// TIA Portal V18 export
// export: Created 2026-06-08T04:47:36.6664765Z, ExportSetting WithDefaults, DisplayName Totally Integrated Automation Portal, DisplayVersion V18, DisplayName TIA Portal Openness, DisplayVersion V18, DisplayName TIA Portal Version Control Interface, DisplayVersion V18, DisplayName STEP 7 Professional, DisplayVersion V18, DisplayName STEP 7 Safety, DisplayVersion V18, DisplayName WinCC Professional, DisplayVersion V18
DATA_BLOCK "MB_SERVER_DB"   // DB53
// stored: AutoNumber true, DBAccessibleFromOPCUA true, InstanceOfName MB_SERVER_3, OfSystemLibElement MB_SERVER, OfSystemLibVersion 3.1
"MB_SERVER_3"
   // VAR_INPUT
   //    DISCONNECT : Bool;
   //    CONNECT_ID : UInt;
   //    IP_PORT : UInt;
   // END_VAR
   // VAR_OUTPUT
   //    NDR : Bool;
   //    DR : Bool;
   //    ERROR : Bool;
   //    STATUS : Word;
   // END_VAR
   // VAR_IN_OUT
   //    MB_HOLD_REG : Variant;
   // END_VAR
   // VAR
   //    TCON_SFB { S7_SetPoint := 'True'} : TCON;
   //    TDISCON_SFB { S7_SetPoint := 'True'} : TDISCON;
   //    TSEND_SFB { S7_SetPoint := 'True'} : TSEND;
   //    TRCV_SFB { S7_SetPoint := 'True'} : TRCV;
   //    TCON_Param { S7_SetPoint := 'True'} : TCON_Param;
   //    MB_State : UInt;
   //    Request_Count : UInt;
   //    Server_Message_Count : UInt;
   //    Xmt_Rcv_Count : UInt;
   //    Exception_Count : UInt;
   //    Success_Count : UInt;
   //    SL_Status_Hold : UInt;
   //    HR_Start_Offset : UInt;
   //    Init_OK : Bool;
   //    SL_Error_State : Bool;
   //    Connected : Bool;
   //    XMT_Set_NDR : Bool;
   //    XMT_Set_DR : Bool;
   // END_VAR
BEGIN
END_DATA_BLOCK
